FUNCTION_BLOCK EL1024
VAR
	_io : EL1xx4_Data;
	{attribute addProperty Name "WcState"}
	_wcState : WcStateInputToggle;
	{attribute addProperty Name "Info data"}
	_infoData : InfoDataBase;
END_VAR

PROPERTY IO : REFERENCE TO EL1xx4_Data
GET
IO REF= _io;
END_GET
END_PROPERTY

PROPERTY WcState : REFERENCE TO WcStateInputToggle
GET
WcState REF= _wcState;
END_GET
END_PROPERTY

END_FUNCTION_BLOCK

(* stored: Version 1.1.0.1, ProductVersion 3.1.4024.9
   POU EL1024: Id {a54687de-07ff-02c8-1b4b-6cb7ccfd3e78}, SpecialFunc None
   Property IO: Id {bc160274-652b-0016-1c71-92ca7d61054a}
   Get Get: Id {0b6bc626-b3d1-079a-2a39-9bfc07b7a3f1}
   Property WcState: Id {b0da1e6f-144d-0e0c-3dba-3afbab11b54b}
   Get Get: Id {fc0539cd-4094-03dd-10cd-a7c3358d9a95} *)
